// TwinCAT 3 PLC project VacProbe
// ProgramVersion: 3.1.4026.16
// libraries:
//   Tc2_SerialCom, * (Beckhoff Automation GmbH)
//   Tc2_Standard, * (Beckhoff Automation GmbH)
//   Tc2_System, * (Beckhoff Automation GmbH)
// project tree:
//   DUTs/ tVacStatus.TcDUT, tRsOut_ITR90.TcDUT
//   / FastTask.TcTTO, PlcTask.TcTTO
//   GVLs/ EL6001.TcGVL
//   POUs/ MAIN.TcPOU, FB_VacSensor.TcPOU, SerialControl.TcPOU
// real-time tasks:
//   TASK PlcTask: cycle T#10ms, priority 20, ADS port 350
//   TASK FastTask: cycle T#1ms, priority 1, ADS port 351
// I/O:
//   DEVICE Device 1 (EtherCAT) (disabled), AmsNetId 10.100.102.11.2.1
//     Term VacMaster (EK1100) [EK1100 EtherCAT Coupler (2A E-Bus)]
//       Term VacAn (EL3072) [EL3072 2Ch. Ana. Input +/-10V, +/-20mA]
//       Term VacRS (EL6001) [EL6001 Interface (RS232)]
// variable links:
//   VacProbe/VacProbe Instance <-> Device 1 (EtherCAT)/Term VacMaster (EK1100)/Term VacAn (EL3072)
//     PlcTask Inputs/MAIN.vacSensor.anStatus <-> AI Standard Channel 1/Status
//     PlcTask Inputs/MAIN.vacSensor.anValue <-> AI Standard Channel 1/Value
//   VacProbe/VacProbe Instance <-> Device 1 (EtherCAT)/Term VacMaster (EK1100)/Term VacRS (EL6001)
//     FastTask Inputs/EL6001.COMin_EL6001_MASTER @bit {16..184 step 8} <-> COM Inputs/Data In {0..21}  (22 links)
//     FastTask Inputs/EL6001.COMin_EL6001_MASTER <-> COM Inputs/Status
//     FastTask Outputs/EL6001.COMout_EL6001_MASTER <-> COM Outputs/Ctrl
//     FastTask Outputs/EL6001.COMout_EL6001_MASTER @bit {16..184 step 8} <-> COM Outputs/Data Out {0..21}  (22 links)

CONFIGURATION VacProbe
    RESOURCE PLC ON TwinCAT3
        TASK FastTask(INTERVAL := T#1ms, PRIORITY := 1);
        TASK PlcTask(INTERVAL := T#10ms, PRIORITY := 20);
        PROGRAM SerialControl WITH FastTask : SerialControl;
        PROGRAM MAIN WITH PlcTask : MAIN;
    END_RESOURCE
END_CONFIGURATION

// ---- DUTs/tVacStatus.TcDUT
TYPE tVacStatus :
STRUCT
	rsBusy         : BOOL := 1;  // RS data not received yet, not an error
	rsErr          : BYTE := 0;
	  
       // bit 0 : No signal for 1sec
       // bit 1 : Pirani adjusted poorly 
	   // bit 2 : BA error 
	   // bit 3 : Pirani error
	   // bit 7 : unknown error code  
	   
	anErr          : BYTE := 0;

       // bit 0 : Underrange  
       // bit 1 : Overrange
       // bit 2 : General error (isn't it just over+underrange? idk)
       // bit 3 : Internal error
END_STRUCT
END_TYPE

// ---- DUTs/tRsOut_ITR90.TcDUT
TYPE tRsOut_ITR90 : ARRAY[1..9] OF byte; END_TYPE

// ---- GVLs/EL6001.TcGVL
{attribute 'qualified_only'}
VAR_GLOBAL
    COMin_EL6001_MASTER AT %I*  : EL6inData22B;
	COMout_EL6001_MASTER AT %Q*  : EL6outData22B;
    RxBuffer_MASTER 			: ComBuffer;
	TxBuffer_MASTER 			: ComBuffer;
	serialCommCtrl              : SerialLineControl;
END_VAR

// ---- POUs/SerialControl.TcPOU
PROGRAM SerialControl
VAR
END_VAR

EL6001.serialCommCtrl(
	Mode := SERIALLINEMODE_EL6_22B,
	pComIn := ADR(EL6001.COMin_EL6001_MASTER),
	SizeComIn := SIZEOF(EL6001.COMin_EL6001_MASTER),
	pComOut := ADR(EL6001.COMout_EL6001_MASTER),
	TxBuffer := EL6001.TxBuffer_MASTER,
	RxBuffer := EL6001.RxBuffer_MASTER);

END_PROGRAM

// ---- POUs/MAIN.TcPOU
PROGRAM MAIN
VAR
	vacSensor : FB_VacSensor;
END_VAR

vacSensor();

END_PROGRAM

// ---- POUs/FB_VacSensor.TcPOU
(* 
  This function block implements double polling of the ITR90 vacuum sensor.
  To retrieve the results, call getValues(RsValue=>, AnValue=>, Status=>):

    RsValue: UINT value from the RS232 output, received via EL6001
    AnValue: UINT value from the analog output, received via EL3072
    Status: data readiness and errors reported; see the tVacStatus type for details

  Error bits in Status reflect all error conditions reported by the sensor, and they accumulate.
  Use clearRsErrors and clearAnErrors functions to reset them.

  Absence of RS232 reports for more than 1 second is also treated as an error.
  Modify RS_TIMEOUT to change the timeout duration.
*)

FUNCTION_BLOCK FB_VacSensor
VAR_INPUT
END_VAR
VAR_OUTPUT
END_VAR
VAR
   fbReceive : ReceiveByte;
   fbReset   : ComReset;
 
   anStatus AT %I* : INT; 
   anValue  AT %I* : INT;
     
     RxSysBuffer : ComBuffer;
   
	 RsWatchdog : TON;
	 
     RsState : INT := 0;
	 RsRecBuffer : tRsOut_ITR90;
	 
	 VacStatus    : tVacStatus;
	 VacAnValue  : UINT := 16#FFFF;
	 VacRsValue  : UINT := 16#FFFF;
	 
   tmrTest : TON;	 
END_VAR
VAR CONSTANT
	 RS_TIMEOUT : TIME := T#1S;	
END_VAR

_readByRs();
_readByAn();

METHOD PRIVATE _readByAn 
VAR_INPUT
END_VAR
IF anStatus.0  THEN VacStatus.anErr.0 := 1; END_IF
IF anStatus.1  THEN VacStatus.anErr.1 := 1; END_IF
IF anStatus.6  THEN VacStatus.anErr.2 := 1; END_IF  
IF anStatus.14 THEN VacStatus.anErr.3 := 1; END_IF
END_METHOD

METHOD PRIVATE _readByRs
VAR_INPUT
END_VAR
VAR
   chksum: INT;
   rsdone : BOOL; 
   rserror : ComError_t;
END_VAR
rsWatchdog(IN := TRUE, PT := RS_TIMEOUT);
IF rsWatchdog.Q THEN VacStatus.rsErr.0 := 1; END_IF 

fbReceive(RxBuffer := RxSysBuffer, 
          ReceivedByte => RsRecBuffer[RsState+1],
          ByteReceived => rsdone, 
	      Error => rserror);

IF NOT (rsdone AND rserror=COMERROR_NOERROR) THEN RETURN; END_IF	

RsState := RsState + 1;
 
CASE RsState OF
	1: IF RsRecBuffer[RsState] <> 7 THEN RsState := 0; END_IF
	2: IF RsRecBuffer[RsState] <> 5 THEN RsState := 0; END_IF
	
	  (* gets bytes 3..8 *)
	
	9: RsState := 0;

	   chksum := RsRecBuffer[2] + RsRecBuffer[3] + RsRecBuffer[4] +
                 RsRecBuffer[5] + RsRecBuffer[6] + RsRecBuffer[7] + RsRecBuffer[8];
   
       IF INT_TO_BYTE(chksum) <> RsRecBuffer[9] THEN RETURN; END_IF

       CASE SHR(RsRecBuffer[4],4) OF
          0: rsWatchdog(IN := FALSE);
             VacStatus.rsBusy := FALSE;  
	      5: VacStatus.rsErr.1 := 1;
	      8: VacStatus.rsErr.2 := 1;
	      9: VacStatus.rsErr.3 := 1;
	   ELSE	 VacStatus.rsErr.7 := 1;
	   END_CASE
	   
       VacRsValue  := RsRecBuffer[6] + SHL(BYTE_TO_UINT(RsRecBuffer[5]),8);
END_CASE
END_METHOD

METHOD clrAnErrors
VAR_INPUT
END_VAR
VacStatus.anErr := 0;
END_METHOD

METHOD clrRsErrors
VAR_INPUT
END_VAR
VacStatus.rsErr  := 0;
VacStatus.rsBusy := TRUE;
rsWatchdog(IN := FALSE);
END_METHOD

METHOD getValues
VAR_INPUT
END_VAR
VAR_OUTPUT
	RsValue : UINT;
	AnValue : UINT;
	Status  : tVacStatus;
END_VAR
Status  := VacStatus;
RsValue := VacRsValue; 
AnValue := VacAnValue;
END_METHOD

END_FUNCTION_BLOCK
